// TIA Portal project "Uygulama 18 (-10V ----  10V)" (V17)

(* hardware
DEVICE "S71500/ET200MP-Station_1"  S7-1500 station
   slot 0: "Profilschiene_0"  6ES7 590-1***0-0AA0
   slot 1: "PLC_1"  CPU 1511-1 PN  6ES7 511-1AK00-0AB0  V1.8
   slot 2: "AI 8xU/I/RTD/TC ST_1"  AI 8xU/I/RTD/TC ST  6ES7 531-7KF00-0AB0  V2.0
   slot 3: "AI 8xU/I/RTD/TC ST_2"  AI 8xU/I/RTD/TC ST  6ES7 531-7KF00-0AB0  V2.0
   slot 4: "AI 8xU/I/RTD/TC ST_3"  AI 8xU/I/RTD/TC ST  6ES7 531-7KF00-0AB0  V2.0
   slot 5: "AI 8xU/I/RTD/TC ST_4"  AI 8xU/I/RTD/TC ST  6ES7 531-7KF00-0AB0  V2.0
   slot 6: "DI 16x24VDC BA_1"  DI 16x24VDC BA  6ES7 521-1BH10-0AA0  V1.0
*)

// ===== PLC "PLC_1"  CPU 1511-1 PN =====

VAR_GLOBAL   // PLC tag table "Standard-Variablentabelle"
   "START" AT %E0.0 : Bool;
   "MOTOR" AT %A0.0 : Bool;
   "STOP" AT %E0.1 : Bool;
   "Tag_1" AT %M0.0 : Bool;
   "Tag_2" AT %I0.2 : Bool;
   "Tag_3" AT %IW30 : Word;
   "Tag_4" AT %MW100 : Word;
   "Tag_5" AT %MW200 : UInt;
   "Tag_6" AT %ID30 : DWord;
   "Tag_7" AT %MD50 : DWord;
   "Tag_8" AT %QD30 : Real;
   "Tag_9" AT %QD34 : DWord;
   "Tag_10" AT %QD38 : DWord;
   "Tag_11" AT %ID34 : DWord;
   "Tag_12" AT %MW55 : Word;
   "Tag_13" AT %MD55 : DWord;
   "Tag_14" AT %IW32 : Word;
   "Tag_15" AT %IW34 : Word;
END_VAR

FUNCTION "MHJ-PLC-Lab-Function-S71500" : Void   // FC9000, SCL
{ S7_Optimized_Access := 'TRUE' }
VERSION : 0.1
   VAR_TEMP
      Value : Byte;
      ForCounter : Int;
   END_VAR
   VAR CONSTANT
      Value_01_DW : DWord := 16#1223_5486;
      Value_02_DW : DWord := 16#A6C9_D1F5;
   END_VAR
BEGIN

   #Value:=PEEK(area := 16#82,
        dbNumber := 0,
        byteOffset := 511);
   #Value := #Value + 1;

   POKE(area := 16#82,
        dbNumber := 0,
        byteOffset := 511,
        value := #Value);

   POKE(area := 16#82,
        dbNumber := 0,
        byteOffset := 1016,
        value := #Value_01_DW);
   POKE(area := 16#82,
        dbNumber := 0,
        byteOffset := 1020,
        value := #Value_02_DW);

   FOR #ForCounter := 0 TO 63 DO
       #Value:=PEEK(area := 16#1,
            dbNumber := 0,
            byteOffset := #ForCounter);
       POKE(area := 16#81,
            dbNumber := 0,
            byteOffset := #ForCounter,
            value := #Value);
   END_FOR;
   #Value := PEEK(area := 16#1,
                  dbNumber := 0,
                  byteOffset := 512);
   POKE(area := 16#82,
        dbNumber := 0,
        byteOffset := 512,
        value := #Value);
END_FUNCTION

ORGANIZATION_BLOCK "Main"   // OB1, LAD, ProgramCycle
TITLE = "Main Program Sweep (Cycle)"
{ S7_Optimized_Access := 'TRUE' }
VERSION : 0.1
   VAR_INPUT
      Initial_Call : Bool;   // Initial call of this OB
      Remanence : Bool;   // =True, if remanent data are available
   END_VAR
BEGIN

REGION Network 1
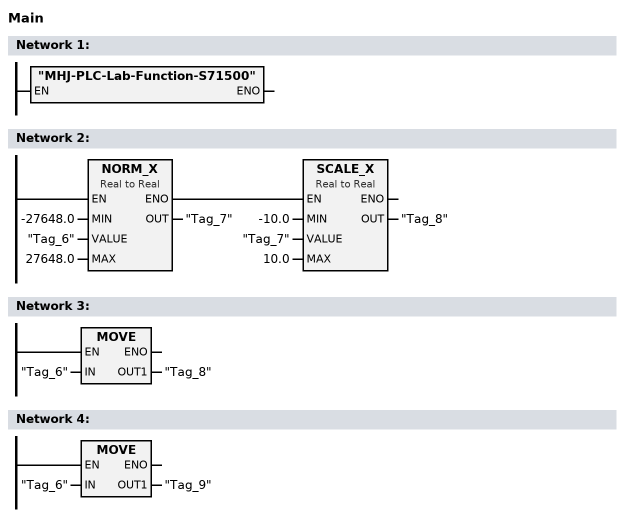
   RUNG wire#powerrail
      "MHJ-PLC-Lab-Function-S71500"()
   END_RUNG
   // the same network as SCL:
   "MHJ-PLC-Lab-Function-S71500"();
END_REGION

REGION Network 2
   RUNG wire#powerrail
      { S7_Templates := "[SrcType := Real, DestType := Real]" } Normalize(min := -27648.0, value := "Tag_6", max := 27648.0, out => "Tag_7")
      { S7_Templates := "[SrcType := Real, DestType := Real]" } Scale(min := -10.0, value := "Tag_7", max := 10.0, out => "Tag_8")
   END_RUNG
   // the same network as SCL:
   "Tag_7" := NORM_X(MIN := -27648.0, VALUE := "Tag_6", MAX := 27648.0);
   "Tag_8" := SCALE_X(MIN := -10.0, VALUE := "Tag_7", MAX := 10.0);
END_REGION

REGION Network 3
   RUNG wire#powerrail
      Move(in := "Tag_6", out1 => "Tag_8")
   END_RUNG
   // the same network as SCL:
   "Tag_8" := "Tag_6";
END_REGION

REGION Network 4
   RUNG wire#powerrail
      Move(in := "Tag_6", out1 => "Tag_9")
   END_RUNG
   // the same network as SCL:
   "Tag_9" := "Tag_6";
END_REGION
END_ORGANIZATION_BLOCK